FUNCTION_BLOCK FB_MotorFreqCtrl
VAR_INPUT
	i_Interlocks		:ARRAY[1..8] OF BOOL;
	i_AutoCmdFwd		:BOOL;
	i_AutoCmdBwd		:BOOL;
	i_AutoSpeedSP		:REAL;
	i_ManCmdFwd			:BOOL;
	i_ManCmdBwd			:BOOL;
	i_ManStop			:BOOL;
	i_ManSpeedSP		:REAL;
	i_Feedback1AP		:REAL;
	i_Feedback2AP		:REAL;
	i_EnableMonitor		:BOOL;
	i_MonitorTime		:INT;
	i_MonitorTolerance	:INT;
	i_ServiceMode		:BOOL;
	i_MaintLimit		:REAL;
	i_PresetValue		:REAL;
	i_WritePreset		:BOOL;
END_VAR
VAR_OUTPUT
	q_InterlocksOK		:BOOL;
	q_bCmdFwd			:BOOL;
	q_bCmdBwd			:BOOL;
	q_SpeedSP			:REAL;
	q_FeedbackMonFlt	:BOOL;
	q_TotalHours		:REAL;
	q_MaintHours		:REAL;
	q_bMaintCall		:BOOL;	
	q_State				:INT;
END_VAR
VAR
	bCmdFwd				:BOOL;
	bCmdBwd				:BOOL;
	tRunTime			:TIME;
	tRunTime1			:TIME;
	rRunTime			:REAL;
	tofCMDFwd			:TOF;
	tofCMDBwd			:TOF;
	tonFwdOff			:TON;
	tonBcwOff			:TON;
	tonMonFdb			:TON;
	tonMotorRun			:TON;
	tofMotorRun			:TOF;
END_VAR
VAR // added by the converter: edge detectors and wires of the graphical bodies
    _w1, _w2 : BOOL;
    _ft1, _ft2 : F_TRIG;
    _rt1 : R_TRIG;
END_VAR

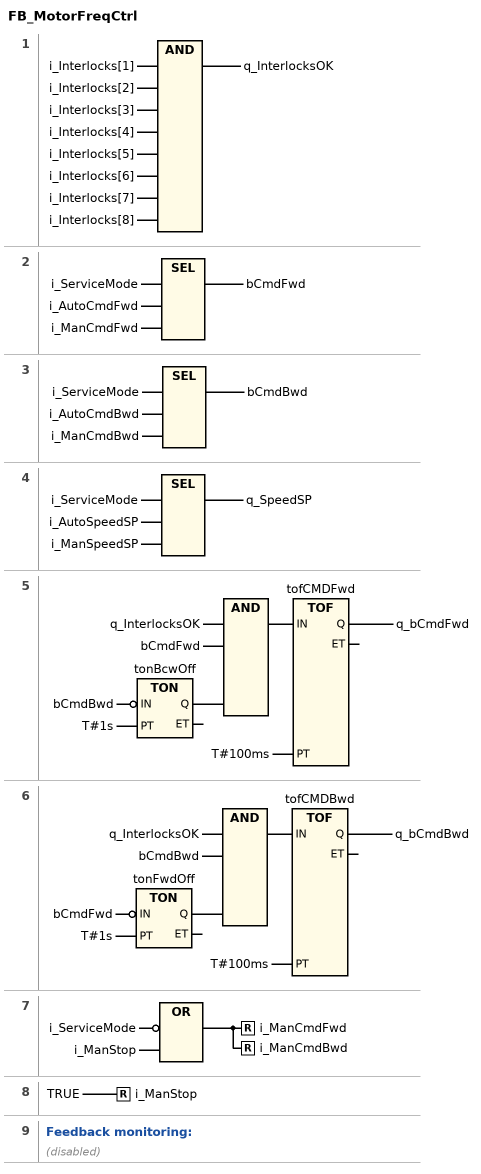
// NETWORK 1
q_InterlocksOK := i_Interlocks[1] AND i_Interlocks[2] AND i_Interlocks[3] AND i_Interlocks[4] AND i_Interlocks[5] AND i_Interlocks[6] AND i_Interlocks[7] AND i_Interlocks[8];

// NETWORK 2
bCmdFwd := SEL(i_ServiceMode, i_AutoCmdFwd, i_ManCmdFwd);

// NETWORK 3
bCmdBwd := SEL(i_ServiceMode, i_AutoCmdBwd, i_ManCmdBwd);

// NETWORK 4
q_SpeedSP := SEL(i_ServiceMode, i_AutoSpeedSP, i_ManSpeedSP);

// NETWORK 5
tonBcwOff(IN := NOT bCmdBwd, PT := T#1s); // TON
tofCMDFwd(IN := q_InterlocksOK AND bCmdFwd AND tonBcwOff.Q, PT := T#100ms); // TOF
q_bCmdFwd := tofCMDFwd.Q;

// NETWORK 6
tonFwdOff(IN := NOT bCmdFwd, PT := T#1s); // TON
tofCMDBwd(IN := q_InterlocksOK AND bCmdBwd AND tonFwdOff.Q, PT := T#100ms); // TOF
q_bCmdBwd := tofCMDBwd.Q;

// NETWORK 7
_w1 := NOT i_ServiceMode OR i_ManStop;
i_ManCmdFwd R= _w1;
i_ManCmdBwd R= _w1;

// NETWORK 8
i_ManStop R= TRUE;

// NETWORK 9 (disabled)
// label: Feedback monitoring

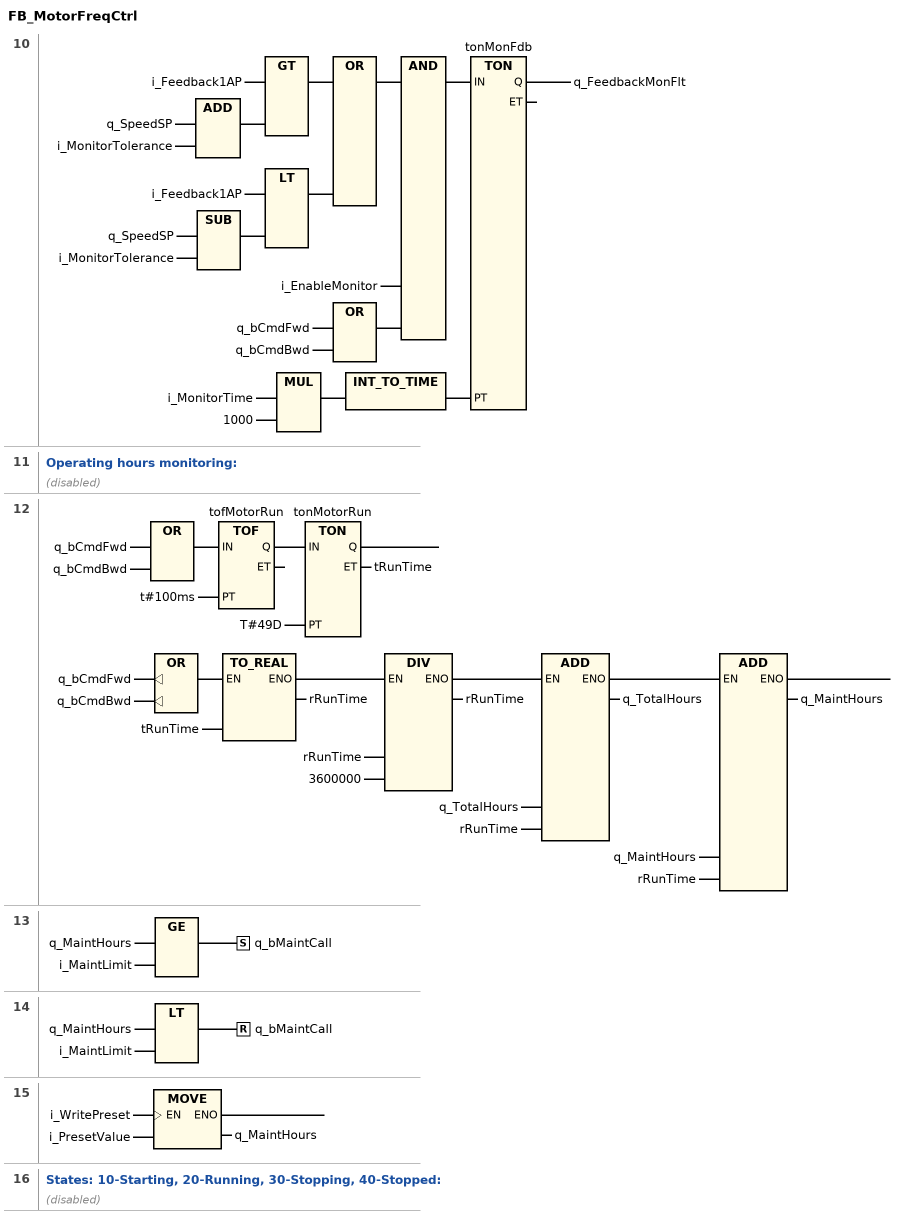
// NETWORK 10
tonMonFdb(IN := (i_Feedback1AP > q_SpeedSP + i_MonitorTolerance OR i_Feedback1AP < q_SpeedSP - i_MonitorTolerance) AND i_EnableMonitor AND (q_bCmdFwd OR q_bCmdBwd), PT := INT_TO_TIME(i_MonitorTime * 1000)); // TON
q_FeedbackMonFlt := tonMonFdb.Q;

// NETWORK 11 (disabled)
// label: Operating hours monitoring

// NETWORK 12
tofMotorRun(IN := q_bCmdFwd OR q_bCmdBwd, PT := t#100ms); // TOF
tonMotorRun(IN := tofMotorRun.Q, PT := T#49D, ET => tRunTime); // TON
_ft1(CLK := q_bCmdFwd);
_ft2(CLK := q_bCmdBwd);
_w2 := _ft1.Q OR _ft2.Q;
IF _w2 THEN rRunTime := TO_REAL(tRunTime); END_IF
IF _w2 THEN rRunTime := rRunTime / 3600000; END_IF
IF _w2 THEN q_TotalHours := q_TotalHours + rRunTime; END_IF
IF _w2 THEN q_MaintHours := q_MaintHours + rRunTime; END_IF

// NETWORK 13
q_bMaintCall S= q_MaintHours >= i_MaintLimit;

// NETWORK 14
q_bMaintCall R= q_MaintHours < i_MaintLimit;

// NETWORK 15
_rt1(CLK := i_WritePreset);
IF _rt1.Q THEN q_MaintHours := i_PresetValue; END_IF

// NETWORK 16 (disabled)
// label: States: 10-Starting, 20-Running, 30-Stopping, 40-Stopped

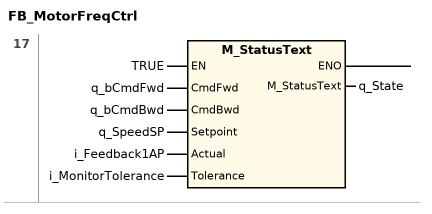
// NETWORK 17
q_State := M_StatusText(CmdFwd := q_bCmdFwd, CmdBwd := q_bCmdBwd, Setpoint := q_SpeedSP, Actual := i_Feedback1AP, Tolerance := i_MonitorTolerance);

METHOD M_StatusText : INT
VAR_INPUT
	CmdFwd		:BOOL;
	CmdBwd		:BOOL;
	Setpoint	:REAL;
	Actual		:REAL;
	Tolerance	:INT;
END_VAR
IF (CmdFwd OR CmdBwd) AND (Actual <= Setpoint-Tolerance+1) THEN
	M_StatusText := 10;	//Starting
ELSIF (CmdFwd OR CmdBwd) AND (Actual >= Setpoint-Tolerance+1) AND (Actual <= Setpoint+Tolerance+1) THEN
	M_StatusText := 20;	//Running
ELSIF (NOT CmdFwd AND NOT CmdBwd) AND (Actual >= 0+Tolerance+1) THEN
	M_StatusText := 30;	//Stopping
ELSIF (NOT CmdFwd AND NOT CmdBwd) AND (Actual <= 0+Tolerance+1)
		OR (NOT CmdFwd AND NOT CmdBwd) AND Setpoint >= Actual THEN
	M_StatusText := 40;	//Stopped
END_IF
END_METHOD

END_FUNCTION_BLOCK

(* stored: Version 1.1.0.1, ProductVersion 3.1.4024.12
   POU FB_MotorFreqCtrl: Id {49f12b5b-7b3f-4962-9afb-5c64de07ca75}, SpecialFunc None
   Method M_StatusText: Id {a49bc4d0-4754-4a54-a919-561375e2ca47} *)
